{attribute 'GeneratedUsingTerminal: EM7004-0000-0017'}
{attribute addProperty BoxType "EM7004-0000-0017"}
{attribute addProperty Id "OutputAT %Q*Output_FFFF807A16"}
{attribute addProperty CRC "1206021482"}
{attribute addProperty Size "16"}
TYPE DO_Outputs_47E26D6A EXTENDS OutputBase_10CEE7DE :
STRUCT
	{attribute addProperty Name "Output"}
	Output AT %Q* : Output_FFFF807A;
END_STRUCT
END_TYPE

(* stored: Version 1.2.0.0, ProductVersion 3.1.4024.11
   DUT DO_Outputs_47E26D6A: Id {8ed838f1-56c3-4d72-8e64-77fe0ad5c67f} *)
